// Brief: Master Arm Cart Control
FUNCTION_BLOCK PUBLIC FB_StateCtrlCart EXTENDS FB_SlaveArmCtrlBase
VAR_INPUT
END_VAR
VAR_OUTPUT
END_VAR
VAR
END_VAR

METHOD PUBLIC init : BOOL
VAR_IN_OUT CONSTANT
	i_slaveArm	:FB_SlaveArm;
END_VAR
VAR_IN_OUT 
	r_slaveArmCtrlCmd :ST_SlaveArmCtrlCmds;
END_VAR

VAR
	j:INT;
	maxJntErr:LREAL;
	jntCtrlErr:Vec7d;
END_VAR
SUPER^.Init(i_slaveArm,r_slaveArmCtrlCmd);

// check if to hold the command joint position unchanged
checkToHoldLastCmds(i_slaveArm,r_slaveArmCtrlCmd);
END_METHOD

END_FUNCTION_BLOCK

(* stored: Version 1.1.0.1, ProductVersion 3.1.4024.12
   POU FB_StateCtrlCart: Id {acf69b98-a94c-45d6-930a-e719a9a02026}, SpecialFunc None
   Method init: Id {4c46dc31-dc49-4fc6-9e65-f4bc803697a8} *)
